// Block: A0201_Profilatrice_RegolazioneFormato_PERS

DATA_BLOCK A0201_Profilatrice_RegolazioneFormato_PERS
VERSION : 0.1
   NON_RETAIN
   VAR
      Par_Machine : Struct
         Passaggio02_MaxDisallineamentoAXs : Real;
         Passaggio14_MaxDisallineamentoAXs : Real;
         Passaggio17_MaxDisallineamentoAXs : Real;
         Passaggio18_MaxDisallineamentoAXs : Real;
         AxD_AutoSpeed : Real;
      END_STRUCT;
      Par_Enc : Array[1..14] of PosFbk_RTN;
      Par_D : Array[1..6] of Positioning_DOL_Machine_Par;
      Par_M : Array[7..14] of Positioning_MOL_Machine_Par;
      Pers_D : Array[1..6] of Positioning_DOL_Machine_Pers_Data;
      Pers_M : Array[7..14] of Positioning_MOL_Machine_Pers_Data;
   END_VAR

BEGIN
   // No initialization required
END_DATA_BLOCK
